TYPE ST_BatchData :
STRUCT
	sBatchID			: STRING;
	sProductionOrder 	: STRING;
	sOperatorID			: STRING;
	sProductItemConfig	: STRING;
	sInputQuantity		: STRING;
END_STRUCT
END_TYPE

(* stored: Version 1.1.0.1, ProductVersion 3.1.4024.9
   DUT ST_BatchData: Id {4b29fe96-cce6-4f26-9ada-3409e2c6c12d} *)
